Fanuc KAREL source: kt00330.KL

PROGRAM KT00330
%STACKSIZE=65535
%PRIORITY=65535
%NOLOCKGROUP
VAR
I1 : INTEGER
R2 : REAL
OUT : BOOLEAN
BEGIN
I1=2
R2=3.0
-- UNSAFE_SOURCE_IR line 10: OUT = (int_to_real(I1) < R2)
END KT00330
